FUNCTION_BLOCK E_MUX_4 (* Event multiplexer (generic FB) *)
  {SET_ATTRIBUTE(eclipse4diac::core::GenericClassName, 'GEN_E_MUX')}
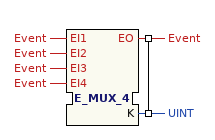
  EVENT_INPUT
    EI1; (* Event to multiplex, K=0 *)
    EI2; (* Event to multiplex, K=1 *)
    EI3; (* Event to multiplex, K=2 *)
    EI4; (* Event to multiplex, K=3 *)
  END_EVENT
  EVENT_OUTPUT
    EO WITH K; (* Event which was multiplexed *)
  END_EVENT
  VAR_OUTPUT
    K : UINT; (* Event index *)
  END_VAR
END_FUNCTION_BLOCK
